% RSLogix 500 project P2_ABIOLA_A_BAK095.RSS, saved by version 8.30.00.16 %
PROJECT "UNTITLED"    % processor: Bul.1763 MicroLogix 1100 Series B %

PROGRAM FILES
  LAD 2   4 rungs
  LAD 3 "INPUT DVS"  1 rungs  % This contains all the input devices used %
  LAD 4 "OUTPUT DVS"  1 rungs  % This contains all the output device used %
  LAD 5 "PRO LOGIC"  1 rungs  % This contains the implementation of the logic %

DATA FILES
  O0 OUTPUT  4 elements
  I1 INPUT  6 elements
  S2 STATUS  66 elements
  B3 BINARY  1 elements
  T4 TIMER  1 elements
  C5 COUNTER  1 elements
  R6 CONTROL  1 elements
  N7 INTEGER  1 elements
  F8 FLOAT  1 elements

LADDER 2
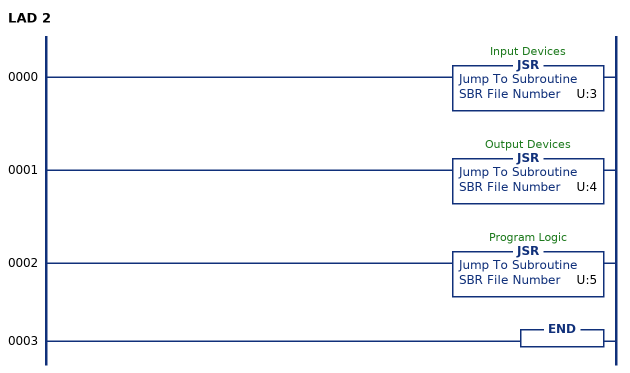
% Rung: 0 %  % edit flag set %
SOR JSR U:3 EOR
%   U:3  "Input Devices" %
% Rung: 1 %  % edit flag set %
SOR JSR U:4 EOR
%   U:4  "Output Devices" %
% Rung: 2 %  % edit flag set %
SOR JSR U:5 EOR
%   U:5  "Program Logic" %
% Rung: 3 %
SOR END EOR
